    # Documented in monorepo/doc/pal/PalAdvancedProgrammingFunctions.md
    def rq_set_conveyor_clearance(is_left_pallet, height):
      if height < 0:
        popup("rq_set_conveyor_clearance(): The clearance height should be positive.", title="Palletizer", error=True,
        blocking=True)
      elif height == 0:
        height = 0.0001
      end

      pallet_side = "right"
      if(is_left_pallet):
         pallet_side = "left"
      end

      local palletId = node_rpc_server.getPalletId(pallet_side)
      node_rpc_server.setConveyorVerticalClearance(palletId, height)
    end
    ###############################################################
    # Linear Axis Move related methods
    ###############################################################
    def verify_is_in_linear_axis_range(target_axis_position):
      axis_position_range = node_rpc_server.linearaxisgetpositionrange()

      if target_axis_position < axis_position_range[0] or target_axis_position > axis_position_range[1]:
        textmsg("Linear axis target position : ", target_axis_position)
        textmsg("Linear axis position range : ", axis_position_range)
        popup("Linear axis position is unreachable.", "Linear Axis Move", blocking=True, error=True)
        halt
      end
    end

    # Documented in monorepo/doc/pal/PalAdvancedProgrammingFunctions.md
    def rq_get_linear_axis_pos():
        axis_position = node_rpc_server.linearaxisgetactualposition()
        return axis_position
    end

  BLOW_OFF_MODE_NO_AIR = 0
  BLOW_OFF_MODE_SMART_AIR = 1
  UNDEFINED_THREAD_ID = -1
  MODBUS_TYPE = "MODBUS"
  STANDARD_TYPE = "STANDARD"
  INVALID_OUTPUT_ADDRESS = -1
  RQ_UNUSED_TIMEOUT = -1

  global rq_cnc_insertion_node_ids = [-1, -1]
  global rq_run_timeout = 30

  ###################################################################################
  #
  # Generic methods
  #
  ###################################################################################

  def bool_to_str(value):
    if value:
      return "true"
    else:
      return "false"
    end
  end

  def bool_array_to_string(array, index):
    if (index >= length(array)):
      return "]"
    end

    separator = ","
    if (index == length(array) - 1):
      separator = ""
    end

    if (index == 0):
      str_array = concat("[", bool_to_str(array[index]), separator)
      return str_cat(str_array, bool_array_to_string(array, index + 1))
    else:
      return concat(bool_to_str(array[index]), separator, bool_array_to_string(array, index + 1))
    end
  end

  def rq_bool_array_to_string(array):
    return bool_array_to_string(array, 0)
  end

  def json_force_node(force, max_negative_deviation, max_positive_deviation, stiffness, enabled_axis, feature, is_adaptive):
    json = "{"
    json = concat(json, key_val("forceFrame", feature), ",")
    json = concat(json, key_val("isAdaptive", is_adaptive), ",")
    json = concat(json, key_val("isForceControlAboutActualPosition", "false"), ",")
    json = concat(json, key_val("isForceMode", enabled_axis), ",")
    json = concat(json, key_val("maxNegativeDeviation", max_negative_deviation), ",")
    json = concat(json, key_val("maxPositiveDeviation", max_positive_deviation), ",")
    json = concat(json, key_val("stiffness", stiffness), ",")
    json = concat(json, key_val("targetTcpWrench", force), "}")
    return json
  end

  def rq_setup_machine_tending_force_node(feature, force, stiffness, max_negative_deviation, max_positive_deviation, enabled_axis, is_adaptive):
    force_node_id = node_rpc_server.createnewforcenode()
    node_rpc_server.fromjson(force_node_id, json_force_node(force, max_negative_deviation, max_positive_deviation,
    stiffness, rq_bool_array_to_string(enabled_axis), 1, bool_to_str(is_adaptive)))
    return force_node_id
  end

  ###################################################################################
  #
  # TRAJECTORY UTILITIES
  #
  ###################################################################################

  def dot_product(v1, v2):
    return [v1]*transpose(v2)
  end

  def get_symmetric_poses_from_middle(p1, p2, middle_pose, distance):
    distance_p1_middle = point_dist(p1, middle_pose)
    alpha = (distance / 2) / distance_p1_middle
    start_pose = interpolate_pose(middle_pose, p1, alpha)
    end_pose = interpolate_pose(middle_pose, p2, alpha)

    return [start_pose, end_pose]
  end

  def translate_to_origin(pose):
    return p[0, 0, 0, pose[3], pose[4], pose[5]]
  end


  ###################################################################################
  #
  # ROBOTIQ PART PRESENTER
  #
  ###################################################################################

  global cnc_part_presenter_index = 0

  def rq_pallet_get_poses_from_index(p_corner_1_approach, p_corners, nb_rows, nb_columns, alternate_direction, index):
      row = floor(index / nb_columns)
      column = index % nb_columns

      row_alpha = 0
      if(nb_rows > 1):
          row_alpha = row / (nb_rows - 1)
      end

      p_row_start = interpolate_pose(p_corners[0], p_corners[3], row_alpha)
      p_row_end = interpolate_pose(p_corners[1], p_corners[2], row_alpha)

      column_alpha = 0
      if(nb_columns > 1):
          column_alpha = column / (nb_columns - 1)
      end

      if(alternate_direction and (row % 2) and nb_columns > 1):
          pallet_pose = interpolate_pose(p_row_end, p_row_start, column_alpha)
      else:
          pallet_pose = interpolate_pose(p_row_start, p_row_end, column_alpha)
      end

      T_1approach_1 = pose_trans(inv(p_corner_1_approach), p_corners[0])
      approach_pose = pose_trans(pallet_pose, inv(T_1approach_1))

      return [approach_pose, pallet_pose]
  end

  ###################################################################################
  #
  # MOVE DOOR
  #
  ###################################################################################

  def rq_setup_door_force_node(reference_frame, force, stiffness):
    feature = 1
    forces = [force,0,0,0,0,0]
    max_negative_deviation = [-5, 0, 0, 0, 0, 0]
    max_positive_deviation = [0.01, 0, 0, 0, 0, 0] # using a large value here would allow the trajectory to violate the kinematics limits, using zero removes the force node effect
    stiffnesses = [stiffness, 100, 100, 100, 100, 100]
    enabled_axis = [True, False, False, False, False, False]
    is_adaptive = True

    force_node_id = rq_setup_machine_tending_force_node(feature, forces, stiffnesses, max_negative_deviation,
    max_positive_deviation, enabled_axis, is_adaptive)

    node_rpc_server.setCustomFixedForceFrame(force_node_id, [reference_frame[3],reference_frame[4],reference_frame[5]])

    return force_node_id
  end

  def json_rq_moves_node(tcp_speed, tcp_accel):
    json = "{"
    json = concat(json, key_val("offsetType", 0), ",")
    json = concat(json, key_val("tcpSpeed", tcp_speed), ",")
    json = concat(json, key_val("tcpAccel", tcp_accel), ",")
    json = concat(json, key_val("actualreferenceframe", [0, 0, 0, 0, 0, 0]), ",")
    json = concat(json, key_val("originalreferenceframe", [0, 0, 0, 0, 0, 0]), "}")
    return json
  end

  def rq_setup_rqmoves_node(parent_node_id, tcp_speed, tcp_accel):
    rq_moves_node_id = node_rpc_server.createnewrqmoves()
    node_rpc_server.fromjson(rq_moves_node_id, json_rq_moves_node(tcp_speed, tcp_accel))
    node_rpc_server.setparentid(rq_moves_node_id, parent_node_id)
    return rq_moves_node_id
  end

  def rq_setup_waypoint_node(pose, joints, is_straight, parent_node_id):
    def json_waypoint_node(pose, joints, is_straight):
      json = "{"
      json = concat(json, key_val("jointPositions", joints), ",")
      json = concat(json, key_val("tcpPose", [pose[0],pose[1],pose[2],pose[3],pose[4],pose[5]]), ",")
      json = concat(json, key_val("isStraight", bool_to_str(is_straight)), "}")
      return json
    end

    waypoint_node_id = node_rpc_server.createnewwaypointnode()
    node_rpc_server.fromjson(waypoint_node_id, json_waypoint_node(pose, joints, is_straight))
    node_rpc_server.setparentid(waypoint_node_id, parent_node_id)
    node_rpc_server.rqmovesaddwaypoint(parent_node_id, waypoint_node_id)
    return waypoint_node_id
  end

  def rq_setup_move_door(reference_frame, start_pose, start_joints, stop_pose, stop_joints, move_force, contact_force, tcp_speed=0.4, tcp_accel=0.4):

    stop_pose_in_start_frame = pose_trans(pose_inv(start_pose), stop_pose)

    seeks_contact = False
    stiffness = 10
    move_force_node_id = rq_setup_door_force_node(reference_frame, move_force, stiffness)
    rq_moves_node_id = rq_setup_rqmoves_node(move_force_node_id, tcp_speed, tcp_accel)
    waypoint_open = rq_setup_waypoint_node(start_pose, start_joints, False, rq_moves_node_id)
    waypoint_close = rq_setup_waypoint_node(stop_pose, stop_joints, True, rq_moves_node_id)
    seeks_contact = True
    stiffness = 100
    contact_force_node_id = rq_setup_door_force_node(reference_frame, contact_force, stiffness)

    rq_movej_node_id = node_rpc_server.createnewmovejnode()
    node_rpc_server.setparentid(rq_movej_node_id, move_force_node_id)

    return [move_force_node_id, rq_moves_node_id, waypoint_open, waypoint_close, contact_force_node_id, rq_movej_node_id]
  end

  def rq_move_door(start_pose, start_joints, stop_pose, stop_joints, move_force, contact_force, tcp_speed, tcp_accel, approach_pose, approach_joints, end_reached_threshold=0.001):

    reference_frame = list_to_pose(kinematics_rpc_server.reorientP1WithXTowardP2andZApproxP1Z(start_pose, stop_pose))

    node_ids = rq_setup_move_door(reference_frame, start_pose, start_joints, stop_pose, stop_joints, move_force, contact_force, tcp_speed, tcp_accel)

    move_force_node_id = node_ids[0]
    rq_moves_node_id = node_ids[1]
    start_waypoint_node_id = node_ids[2]
    end_waypoint_node_id = node_ids[3]
    contact_force_node_id = node_ids[4]
    rq_movej_node_id = node_ids[5]

    rq_wait_ft_sensor_steady(2000)
    zero_ftsensor()
    sleep(0.1)

    path_answer = node_rpc_server.rqmovesinit(rq_moves_node_id)
    verify_path_answer(path_answer)

    approach_position_joints = get_inverse_kin(approach_pose, qnear=approach_joints)
    movej(approach_position_joints)

    node_rpc_server.movejdefinewaypoint(rq_movej_node_id, get_actual_joint_positions(), 1.0, 1.0)
    node_rpc_server.setparentid(rq_movej_node_id, move_force_node_id)
    reset_node_executor()
    active_and_reset_node(move_force_node_id)
    node_execution_thread = execute_node(rq_movej_node_id, True)

    path_answer = node_rpc_server.rqmovesinit(rq_moves_node_id)
    verify_path_answer(path_answer)
    q0 = node_rpc_server.rqmovesgetfirstpoint(rq_moves_node_id)
    node_rpc_server.setparentid(rq_movej_node_id, move_force_node_id)
    node_rpc_server.movejdefinewaypoint(rq_movej_node_id, q0, 1.0, 0.4)
    execute_node(rq_movej_node_id)
    execute_node(start_waypoint_node_id)
    execute_node(end_waypoint_node_id)

    kill_thread(node_execution_thread)

    node_rpc_server.movejdefinewaypoint(rq_movej_node_id, get_actual_joint_positions(), 1.0, 1.0)
    node_rpc_server.setparentid(rq_movej_node_id, contact_force_node_id)
    reset_node_executor()
    active_and_reset_node(contact_force_node_id)
    node_execution_thread = execute_node(rq_movej_node_id, True)

    timeout = 20
    while (point_dist(get_actual_tcp_pose(), stop_pose) > end_reached_threshold):
      if (timeout <= 0):
        popup("Door has not reached its final position")
        halt
      else:
        sync()
        timeout = timeout - get_steptime()
      end
    end

    kill_thread(node_execution_thread)

    approach_pose_in_start_frame = pose_trans(pose_inv(start_pose), approach_pose)
    retract_pose = pose_trans(get_actual_tcp_pose(), approach_pose_in_start_frame)
    movej(retract_pose)

    node_rpc_server.deletenode(move_force_node_id)
    node_rpc_server.deletenode(rq_moves_node_id)
    node_rpc_server.deletenode(start_waypoint_node_id)
    node_rpc_server.deletenode(end_waypoint_node_id)
    node_rpc_server.deletenode(contact_force_node_id)
    node_rpc_server.deletenode(rq_movej_node_id)

  end

  ###################################################################################
  #
  # CNC Insertion
  #
  ###################################################################################

  def rq_collet_insertion(contact_pose, insert_pose, inserted_pose):
      movel(contact_pose, a=1.2, v=0.025)
      movel(insert_pose, a=1.2, v=0.025)

      zero_ftsensor()
      sleep(0.1)

      direction = "Z+"
      stop_force_threshold = 3.0
      max_radius = 5.0
      radius_incr = 0.7
      peck_mode = False
      tangential_speed = 0.02
      compliant_insert_force_threshold = 10.0
      spiral_initial_pose_offset_name = "spiral_initial_pose_offset_name"
      rq_ins_destination = inserted_pose
      max_distance = point_dist(inserted_pose, get_actual_tcp_pose())
      rq_spiral_not_completed = False
      rq_ins_speed_setting = 0.02

      rq_insert_spiral_urcap(direction, stop_force_threshold, max_radius, radius_incr, peck_mode, tangential_speed, compliant_insert_force_threshold, spiral_initial_pose_offset_name)

      if (rq_spiral_not_completed):
        return False
      end

      return True
  end

  def rq_push_part(approach_pose, chuck_pose):
      zero_ftsensor()
      sleep(0.1)

      # Find pose with z axis pointing in the direction of the insertion
      p1 = translate_to_origin(approach_pose)
      insertion_dir_in_base_frame = pose_trans(p1, pose_trans(pose_inv(approach_pose), chuck_pose))
      ref_frame_pose = list_to_pose(kinematics_rpc_server.poseFromZaxis([insertion_dir_in_base_frame[0], insertion_dir_in_base_frame[1], insertion_dir_in_base_frame[2]]))

      surface_found = rq_linear_search_custom_frame("Z+", 10.0, 0.025, 0.1, ref_frame_pose)

      if not(surface_found):
          return False
      end

      return True
  end

  def rq_place_in_chuck(close_chuck_do, open_chuck_do, chuck_approach, chuck_position, chuck_delay):
      rq_open_workholding(close_chuck_do, open_chuck_do)

      movel(chuck_approach, a=1.2, v=0.25)
      movel(chuck_position, a=1.2, v=0.25)

      rq_close_workholding(close_chuck_do, open_chuck_do)
      sleep(chuck_delay)
  end

  def rq_pre_pick_in_chuck(chuck_approach, chuck_position, speed=0.25, accel=1.2):
      movel(chuck_approach, accel, speed)
      movel(chuck_position, accel, speed)
  end

  def rq_post_pick_in_chuck(close_chuck_do, open_chuck_do, chuck_approach, chuck_position, chuck_delay, speed=0.25,
  accel=1.2):
      rq_open_workholding(close_chuck_do, open_chuck_do)
      sleep(chuck_delay)

      movel(chuck_approach, accel, speed)
  end

  def rq_open_workholding(close_do, open_do):
      rq_set_workholding_do(close_do, open_do, False)
  end

  def rq_close_workholding(close_do, open_do):
      rq_set_workholding_do(close_do, open_do, True)
  end

  def rq_set_workholding_do(close_do, open_do, close_request):
      is_close_do_valid = rq_is_do_valid(close_do)
      is_open_do_valid = rq_is_do_valid(open_do)

      if(is_close_do_valid):
          set_standard_digital_out(close_do, close_request)
      end
      if(is_open_do_valid):
          set_standard_digital_out(open_do, not close_request)
      end
      if(is_close_do_valid or is_open_do_valid):
          sleep(0.5)
      end
  end

  def rq_is_do_valid(do_id):
      return do_id >= 0 and do_id <= 7
  end

  def set_cleaning_digital_output(address, state, blow_off_mode, output_type):
     if(blow_off_mode == BLOW_OFF_MODE_SMART_AIR):
       rq_set_output(output_type, address, state)
     end
  end

  ###################################################################################
  #
  # PATH GENERATOR 6 POINTS CURVE BUILT WITH 2 POINTS
  #
  ###################################################################################

  def execute_half_pipe(pose_1, pose_2,pose_transformation_air_nozzle_to_actual_tcp, depth, length_distance, width, angle, speed, spacing, address, output_type, blow_off_mode, passes):
    path_gen_poses = get_path_generator_6_points_poses(pose_1, pose_2, pose_transformation_air_nozzle_to_actual_tcp, depth, length_distance, width, angle)
    start_pose = p[path_gen_poses[0,0],path_gen_poses[0,1],path_gen_poses[0,2],path_gen_poses[0,3],path_gen_poses[0,4],path_gen_poses[0,5]]
    path_generator_node_id = setup_path_generator_6_points(path_gen_poses, speed, spacing)
    execute_path_generator_6_points(path_generator_node_id, start_pose,  address, output_type, blow_off_mode, passes)
  end

  def get_path_generator_6_points_poses(pose_2, pose_5,pose_transformation_air_nozzle_to_actual_tcp, depth=0.01, length=0, width=0.05, angle_deg=0):

    def offset_pose(pose, offset, offset_reference_frame, pose_transformation_air_nozzle_to_actual_tcp):
      pose_relative_to_ref_frame = express_pose_A_relative_to_pose_B(pose, offset_reference_frame)
      ref_frame_with_offset = pose_trans(offset_reference_frame, offset)
      pose_with_offset = pose_trans(ref_frame_with_offset, pose_relative_to_ref_frame)
      pose_with_offset_for_actual_tcp = pose_trans(pose_with_offset, pose_transformation_air_nozzle_to_actual_tcp)
      return pose_to_list(pose_with_offset_for_actual_tcp)
    end

    if(length > 0):
      middle_pose = interpolate_pose(pose_2, pose_5, 0.5)

      poses = get_symmetric_poses_from_middle(pose_2, pose_5, middle_pose, length)
      pose_2 = poses[0]
      pose_5 = poses[1]
    end

    path_ref_frame = list_to_pose(kinematics_rpc_server.reorientP1WithXTowardP2andZApproxP1Z(pose_2, pose_5))

    offset1 = pose_add(p[0,0,0,0,d2r(angle_deg),0], p[0, width,-depth,-d2r(angle_deg),0,0])
    offset2 = pose_add(p[0,0,0,0,d2r(angle_deg),0], p[0,     0,     0,              0,0,0])
    offset3 = pose_add(p[0,0,0,0,d2r(angle_deg),0], p[0,-width,-depth, d2r(angle_deg),0,0])

    pose_1_array = offset_pose(pose_2, offset1, path_ref_frame, pose_transformation_air_nozzle_to_actual_tcp)
    pose_2_array = offset_pose(pose_2, offset2, path_ref_frame, pose_transformation_air_nozzle_to_actual_tcp)
    pose_3_array = offset_pose(pose_2, offset3, path_ref_frame, pose_transformation_air_nozzle_to_actual_tcp)

    pose_4_array = offset_pose(pose_5, offset1, path_ref_frame, pose_transformation_air_nozzle_to_actual_tcp)
    pose_5_array = offset_pose(pose_5, offset2, path_ref_frame, pose_transformation_air_nozzle_to_actual_tcp)
    pose_6_array = offset_pose(pose_5, offset3, path_ref_frame, pose_transformation_air_nozzle_to_actual_tcp)

    return [pose_1_array, pose_2_array, pose_3_array, pose_4_array, pose_5_array, pose_6_array]
  end

  def setup_path_generator_6_points(pose_list, tcp_speed=0.1, spacing=0.02):

    def json_path_generator_node(pose_list, tcp_speed, spacing):

      SIX_POINTS_CURVE = 3
      OFFSET_TYPE_NONE = 0
      FORCE_OPPOSITE_SIDE = 2

      json = "{"
      json = concat(json, key_val("tcpSpeed", tcp_speed), ",")
      json = concat(json, key_val("poses", pose_list), ",")
      json = concat(json, key_val("avoidAbruptEnd", "false"), ",")
      json = concat(json, key_val("isSurfaceFillOn", "true"), ",")
      json = concat(json, key_val("spacing", spacing), ",")
      json = concat(json, key_val("pathType", SIX_POINTS_CURVE), ",")
      json = concat(json, key_val("offsetType",OFFSET_TYPE_NONE), ",")
      json = concat(json, key_val("endingMode", FORCE_OPPOSITE_SIDE), "}")

      return json
    end

    rq_path_generator_parent_id = 0
    path_generator_node_id = node_rpc_server.createPathGeneratorNode()
    node_rpc_server.fromjson(path_generator_node_id, json_path_generator_node(pose_list, tcp_speed, spacing))
    node_rpc_server.setparentid(path_generator_node_id, rq_path_generator_parent_id)

    return path_generator_node_id
  end

  def execute_path_generator_6_points(path_generator_node_id, pose_1, address = INVALID_OUTPUT_ADDRESS, output_type = MODBUS_TYPE, blow_off_mode = BLOW_OFF_MODE_NO_AIR, passes = 1):
    index = 0
    while (index < passes):
      movej(get_inverse_kin(pose_1))
      set_cleaning_digital_output(address, True, blow_off_mode, output_type)
      reset_node_executor()
      node_execution_thread = execute_node(path_generator_node_id, True)
      rq_continue_node_execution = False
      set_cleaning_digital_output(address, False, blow_off_mode, output_type)
      join node_execution_thread
      index = index + 1
    end
    node_rpc_server.deletenode(path_generator_node_id)
  end

  ###################################################################################
  #
  # Straight line trajectory
  #
  ###################################################################################

  def execute_straight_line(p1, p2,pose_transformation_air_nozzle_to_actual_tcp, accel=1.2, speed=0.25, distance = 0, angles = [0, 0, 0], address = INVALID_OUTPUT_ADDRESS, output_type = MODBUS_TYPE, blow_off_mode = BLOW_OFF_MODE_NO_AIR, passes = 1):
    offset_for_angles = p[0, 0, 0, d2r(angles[0]), d2r(angles[1]), d2r(angles[2])]
    p1 = pose_trans(p1, offset_for_angles)
    p2 = pose_trans(p2, offset_for_angles)

    # apply transformation to take into account that the actual tcp offset is not the same as the one that was used when the waypoints were saved:
    p1 = pose_trans(p1, pose_transformation_air_nozzle_to_actual_tcp)
    p2 = pose_trans(p2, pose_transformation_air_nozzle_to_actual_tcp)
    global air_output_adress = address

    qActual = get_actual_joint_positions()
    CleanPathId = node_rpc_server.createnewcleaningpathnode(p1, p2, qActual, passes, distance, accel, speed, blow_off_mode)

    reset_node_executor()
    if output_type == MODBUS_TYPE:
      air_thread = run modbusAirControlThread()
    elif output_type == STANDARD_TYPE:
      air_thread = run standardAirControlThread()
    end

    node_execution_thread = execute_node(CleanPathId, True)
    rq_continue_node_execution = False

    join node_execution_thread
    node_rpc_server.deletenode(CleanPathId)
    if output_type == MODBUS_TYPE or output_type == STANDARD_TYPE :
      kill air_thread
    end
  end

  ###################################################################################
  #
  # Cross trajectory
  #
  ###################################################################################

  def find_cross_trajectory_poses(p1, p2, height=0, width=0, p1_angles = [0, 0, 0], p2_angles = [0, 0, 0], p3_angles = [0, 0, 0], p4_angles = [0, 0, 0]):
    def find_side_poses(p0, p1):
      def find_side_pose(p0,p1,angle):
        p1_T_p0 = pose_trans(pose_inv(p0), p1)
        rotated_p0_by_90_degrees = pose_trans(p0, p[0, 0, 0, 0, 0, d2r(angle)])

        side_pose = pose_trans(rotated_p0_by_90_degrees, p1_T_p0)
        side_pose[3] = p0[3]
        side_pose[4] = p0[4]
        side_pose[5] = p0[5]

        return side_pose
      end

      p3= find_side_pose(p0, p1, 90)
      p4 = find_side_pose(p0, p1, 270)

      return [p3, p4]
    end

    def get_start_and_end_poses_based_on_distance(p1, p2, middle_pose, distance):
      if(distance == 0):
        start_pose = p1
        end_pose = p2
      else:
        poses = get_symmetric_poses_from_middle(p1, p2, middle_pose, distance)
        start_pose = poses[0]
        end_pose = poses[1]
      end
      return [start_pose, end_pose]
    end

    def get_side_poses_based_on_distance(p1, p2, middle_pose, width):
      if(width == 0):
        side_poses = find_side_poses(middle_pose, p1)
      else:
        poses = get_symmetric_poses_from_middle(p1, p2, middle_pose, width)
        side_poses = find_side_poses(middle_pose, poses[0])
      end

      return side_poses
    end

    def get_angle_offset(angles):
      return  p[0, 0, 0, d2r(angles[0]), d2r(angles[1]), d2r(angles[2])]
    end

    middle_pose = interpolate_pose(p1, p2, 0.5)

    start_and_end_poses = get_start_and_end_poses_based_on_distance(p1, p2, middle_pose, height)
    side_poses = get_side_poses_based_on_distance(p1, p2, middle_pose, width)

    p1_offset = get_angle_offset(p1_angles)
    p2_offset = get_angle_offset(p2_angles)
    p3_offset = get_angle_offset(p3_angles)
    p4_offset = get_angle_offset(p4_angles)

    start_and_end_poses[0] = pose_trans(start_and_end_poses[0], p1_offset)
    start_and_end_poses[1] = pose_trans(start_and_end_poses[1], p2_offset)
    side_poses[0] = pose_trans(side_poses[0], p3_offset)
    side_poses[1] = pose_trans(side_poses[1], p4_offset)

    return [middle_pose, start_and_end_poses[0], start_and_end_poses[1], side_poses[0], side_poses[1]]
  end

  def execute_cross_trajectory(p1, p2,pose_transformation_air_nozzle_to_actual_tcp, height=0, width=0, p1_angles = [0, 0, 0], p2_angles = [0, 0, 0], p3_angles = [0, 0, 0], p4_angles = [0, 0, 0], accel=1.2, speed=0.25,  address = INVALID_OUTPUT_ADDRESS, output_type = MODBUS_TYPE, blow_off_mode = BLOW_OFF_MODE_NO_AIR, passes = 1):

    cross_poses = find_cross_trajectory_poses(p1, p2, height, width, p1_angles, p2_angles, p3_angles, p4_angles)

    p0 = pose_trans(cross_poses[0], pose_transformation_air_nozzle_to_actual_tcp)
    p1 = pose_trans(cross_poses[1], pose_transformation_air_nozzle_to_actual_tcp)
    p2 = pose_trans(cross_poses[2], pose_transformation_air_nozzle_to_actual_tcp)
    p3 = pose_trans(cross_poses[3], pose_transformation_air_nozzle_to_actual_tcp)
    p4 = pose_trans(cross_poses[4], pose_transformation_air_nozzle_to_actual_tcp)

   index = 0

   while (index < passes):
     movej(get_inverse_kin(p0))
     set_cleaning_digital_output(address, True, blow_off_mode, output_type)
     movel(p1, accel, speed)
     movel(p2, accel, speed)
     movel(p0, accel, speed)
     movel(p3, accel, speed)
     movel(p4, accel, speed)
     set_cleaning_digital_output(address, False, blow_off_mode, output_type)
     index = index + 1
   end
  end

  def execute_waypoint_cross_trajectory(starting_pose, finishing_pose, accel=1.2, speed=0.25):
   movej(get_inverse_kin(starting_pose))
   movel(finishing_pose, accel, speed)
  end

  ###################################################################################
  #
  # Fermat spiral trajectory
  #
  ###################################################################################

  def execute_fermat_spiral(start_pose, end_pose,pose_transformation_air_nozzle_to_actual_tcp, max_radius = 0, angle = 0, number_of_turns = 1, speed = 0.25,address = INVALID_OUTPUT_ADDRESS, output_type = MODBUS_TYPE, blow_off_mode = BLOW_OFF_MODE_NO_AIR, passes = 1):
    def find_middle(start_pose, end_pose):
      alpha = 0.5
      return interpolate_pose(start_pose, end_pose, alpha)
    end

    def find_next_theta(spiral_constant, theta, speed):
      denom = spiral_constant * sqrt(1/(4*theta) + theta)
      theta_dot = speed / denom
      theta = theta + theta_dot * rq_controller_time_step
      return theta
    end

    def find_spiral_pose(theta, spiral_plane, center_pose, angle, spiral_constant, pose_transformation_air_nozzle_to_actual_tcp):
      local r = spiral_constant * sqrt(theta)
      local x = r * cos(theta)
      local y = r * sin(theta)

      local p2 = pose_trans(spiral_plane, p[x,y,0,0,0,0])
      local p3 = p[p2[0], p2[1], p2[2], center_pose[3], center_pose[4], center_pose[5]]
      local p4 = pose_trans(p3, pose_transformation_air_nozzle_to_actual_tcp)
      local p5 = pose_trans(p4, p[0, 0, 0, -d2r(angle)*cos(theta), -d2r(angle)*sin(theta), 0])
      return p5
    end

    def execute_outer_to_inner_spiral(start_pose, middle_pose, spiral_plane, pose_transformation_air_nozzle_to_actual_tcp, max_angle, angle, spiral_constant_nominal, speed, address, output_type, blow_off_mode):
      local theta = max_angle
      local max_r = point_dist(start_pose, middle_pose)
      local spiral_constant = -1 * spiral_constant_nominal
      local r = max_r
      local is_first_pose = True

      while (norm((r)) <= max_r):
        theta = find_next_theta(spiral_constant, theta, speed)
        if(theta < 0):
          break
        end

        r = spiral_constant * sqrt(theta)
        next_pose = find_spiral_pose(theta, spiral_plane, middle_pose, angle, spiral_constant, pose_transformation_air_nozzle_to_actual_tcp)

        if (is_first_pose):
          movej(get_inverse_kin(next_pose))
          set_cleaning_digital_output(address, True, blow_off_mode, output_type)
          is_first_pose = False
        else:
          servoj(get_inverse_kin(next_pose), t = rq_controller_time_step)
        end
      end
    end

    def execute_inner_to_outer_spiral(start_pose, middle_pose, spiral_plane, pose_transformation_air_nozzle_to_actual_tcp, angle, spiral_constant, speed):
      local theta = 0.0001
      local max_r = point_dist(start_pose, middle_pose)
      local r = 0

      while (norm(r) <= max_r):
        theta = find_next_theta(spiral_constant, theta, speed)
        r = spiral_constant * sqrt(theta)
        next_pose = find_spiral_pose(theta, spiral_plane, middle_pose, angle, spiral_constant, pose_transformation_air_nozzle_to_actual_tcp)
        servoj(get_inverse_kin(next_pose), t = rq_controller_time_step)
      end
    end

    max_angle = d2r(number_of_turns * 360)
    middle_pose = find_middle(start_pose, end_pose)

    if(max_radius > 0):
      poses = get_symmetric_poses_from_middle(start_pose, end_pose, middle_pose, max_radius * 2)
      start_pose = poses[0]
      end_pose = poses[1]
    end

    SPIRAL_CONSTANT = (point_dist(middle_pose, start_pose)) / sqrt(max_angle)

    spiral_plane = list_to_pose(kinematics_rpc_server.reorientP1WithXTowardP2andZApproxP1Z(middle_pose, end_pose))


    index = 0
    while(index < passes):
      execute_outer_to_inner_spiral(start_pose, middle_pose, spiral_plane,pose_transformation_air_nozzle_to_actual_tcp, max_angle, angle, SPIRAL_CONSTANT, speed, address, output_type, blow_off_mode)
      execute_inner_to_outer_spiral(end_pose, middle_pose, spiral_plane, pose_transformation_air_nozzle_to_actual_tcp, angle, SPIRAL_CONSTANT, speed)
      set_cleaning_digital_output(address, False, blow_off_mode, output_type)
      index = index + 1
    end
  end

  ###################################################################################
  #
  # ROBOTIQ VISE INSERTION
  #
  # - The first touch is performed in the direction of the gravity, regardless of
  #   the robot mounting orientation, tcp offset and TCP orientation
  # - Optional 2e et 3e touch are performed relative to TCP. They require that, at
  #   the moment that the insertion is performed, the TCP is oriented such that one
  #   axis is aligned with the gravity. The TCP axes for the 2e and 3e touch are
  #   chosen as the ones not aligned with the gravity.
  ###################################################################################
  def insert_in_vise(start_pose, end_pose, number_of_touch=3, forces=[10, 20, 20], invert_axis=False, move_to_end_pose=False):

    def list_by_scalar_multiply_(l1, scalar):
      result = l1
      i=0
      while i<length(result):
        result[i]=l1[i]*scalar
        i=i+1
      end
      return result
    end

    def find_gravity_direction(acceleration_direction, threshold):
      result = [False, False, False]
      i = 0
      while i < length(result):
        result[i] =  norm(acceleration_direction[i]) > threshold
        i = i + 1
      end
      return result
    end

    def get_axis(index, direction):
      axis = "XYZ"
      if direction < 0:
        sign = "-"
      elif direction > 0:
        sign = "+"
      else:
        popup("insert_in_vise:get_axis >>> direction cannot be 0. Fix it.")
        halt
      end
      return str_cat(str_sub(axis, index, 1), sign)
    end

    def direction_to_index(str):
      if "X" == str_sub(str, 0, 1):
        return 0
      elif "Y" == str_sub(str, 0, 1):
        return 1
      elif "Z" == str_sub(str, 0, 1):
        return 2
      else:
        popup("invalid direction :", str)
        halt
      end
    end

    def find_touch_direction(mask, direction):
      i = 0
      result = [0, 0, 0]
      while i < 3:
        if mask[i]:
          result[i] = direction[i]
        end
        i = i + 1
      end
      return result
    end

    def find_touch_direction_str(mask, direction):
      i = 0
      result = ""
      while i < 3:
        if mask[i]:
          result = str_cat(result, get_axis(i, direction[i]))
        end
        i = i + 1
      end
      return result
    end

    def invert(list):
      result = list
      i = 0
      while i < length(list):
        result[i] = not list[i]
        i = i + 1
      end
      return result
    end

    def assert_that_the_first_touch_is_aligned_with_an_axis(first_touch_direction_mask):
      i = 0
      counter = 0
      while i < length(first_touch_direction_mask):
        if first_touch_direction_mask[i]:
          counter = counter + 1
        end
        i = i + 1
      end

      if counter != 1:
        popup("One of the TCP axes must be perpendicular to the floor while loading the part in the vise.")
        halt
      end
    end

    def setup_nodes(forces, number_of_touch, first_touch_direction_mask, direction, second_direction_str, third_direction_str):
      def max_deviation_from(forces, enabled_axis):
        i = 0
        deviation = [0, 0, 0, 0, 0, 0]
        while i < 3:
          if forces[i] > 0:
            deviation[i] = 10
          elif forces[i] ==  0:
            deviation[i] = 10
          end
          i = i + 1
        end
        while i < 6:
          if enabled_axis[i]:
            deviation[i] = 0.35
          end
          i = i + 1
        end
        return deviation
      end

      def min_deviation_from(forces, enabled_axis):
        i = 0
        deviation = [0, 0, 0, 0, 0, 0]
        while i < 3:
          if forces[i] < 0:
            deviation[i] = -10
          elif forces[i] ==  0:
            deviation[i] = -10
          end
          i = i + 1
        end
        while i < 6:
          if enabled_axis[i]:
            deviation[i] = -0.35
          end
          i = i + 1
        end
        return deviation
      end

      def stiffness_from(forces):
        i = 0
        stiffness = [0, 0, 0, 100, 100, 100]
        while i < length(forces):
          if norm(forces[i]) > 0:
            stiffness[i] = 100
          else:
            stiffness[i] = 85
          end
          i = i + 1
        end
        return stiffness
      end

      def compute_final_forces(forces, number_of_touch, first_touch_direction_mask, direction, second_direction_str, third_direction_str):
        final_forces = [0, 0, 0]
        if number_of_touch > 0:
          i = 0
          while i < length(first_touch_direction_mask):
            if first_touch_direction_mask[i]:
              break
            end
            i = i + 1
          end
          final_forces[i] = direction[i] * forces[i]
        end
        if number_of_touch > 1:
          i = direction_to_index(second_direction_str)
          final_forces[i] = direction[i] * forces[i]
        end
        if number_of_touch > 2:
          i = direction_to_index(third_direction_str)
          final_forces[i] = direction[i] * forces[i]
        end
        return final_forces
      end

      def compute_enabled_axis(first_touch_direction_mask):
        enabled_axis = [True, True, True, False, False, False]
        i = 0
        while i < length(first_touch_direction_mask):
          if first_touch_direction_mask[i]:
            break
          end
          i = i + 1
        end
        enabled_axis[i + 3] = True

        return enabled_axis
      end

      final_forces = compute_final_forces(forces, number_of_touch, first_touch_direction_mask, direction, second_direction_str, third_direction_str)
      enabled_axis = compute_enabled_axis(first_touch_direction_mask)

      force_node_id = rq_setup_machine_tending_force_node(1, [final_forces[0], final_forces[1], final_forces[2], 0, 0, 0], stiffness_from
      (final_forces), min_deviation_from(final_forces, enabled_axis), max_deviation_from(final_forces, enabled_axis),
      enabled_axis, False)
      movej_node_id = node_rpc_server.createnewmovejnode()
      node_rpc_server.setparentid(movej_node_id, force_node_id)

      return [force_node_id, movej_node_id]
    end

    def average_tool_acceleration_reading(n_samples, delay):
      n = n_samples
      reading = [0, 0, 0]
      while n > 0:
        reading = reading + get_tool_accelerometer_reading()
        sleep(delay)
        n = n - 1
      end
      return reading/n_samples
    end

    def linear_search_toward_gravity(force):
      # maybe add a stopj here to prevent acceleration reading to be influenced by robot movement
      flange_accel = average_tool_acceleration_reading(10, 0.1) # measured accel is oriented in gravity oposite direction
      flange_accel_pose = p[-flange_accel[0], -flange_accel[1], -flange_accel[2], 0, 0,0]
      p1 = translate_to_origin(get_actual_tool_flange_pose())
      gravity_dir_in_base_frame = pose_trans(p1, flange_accel_pose)

      # Find pose with z axis pointing in gravity direction:
      ref_frame_pose = list_to_pose(kinematics_rpc_server.poseFromZaxis([gravity_dir_in_base_frame[0], gravity_dir_in_base_frame[1], gravity_dir_in_base_frame[2]]))
      speed = 0.01
      abs_max_distance = 0.05

      surface_found = rq_linear_search_custom_frame("Z+", force, speed, abs_max_distance, ref_frame_pose)
      return surface_found
    end

    #### Actual insert_in_vise method ####
    movel(start_pose)
    zero_ftsensor()

    # 1. Use accelerometer reading to find touches directions:
    ACCELERATION_THRESHOLD = 8
    flange_accel = average_tool_acceleration_reading(10, 0.1)
    tcp_accel = pose_trans(pose_inv(get_tcp_offset()), p[flange_accel[0], flange_accel[1], flange_accel[2], 0, 0, 0])
    first_touch_direction_mask = find_gravity_direction(tcp_accel, ACCELERATION_THRESHOLD)
    assert_that_the_first_touch_is_aligned_with_an_axis(first_touch_direction_mask)

    direction_transform = pose_trans(pose_inv(start_pose), end_pose)
    direction = [direction_transform[0], direction_transform[1], direction_transform[2]]
    direction_sign = [direction[0]/norm(direction[0]), direction[1]/norm(direction[1]), direction[2]/norm(direction[2])]

    touch_direction_str = find_touch_direction_str(invert(first_touch_direction_mask), direction_sign)
    touch_direction = find_touch_direction(invert(first_touch_direction_mask), direction_sign)

    if invert_axis:
      second_direction_str = str_sub(touch_direction_str, 0, 2)
      third_direction_str = str_sub(touch_direction_str, 2, 4)
    else:
      second_direction_str = str_sub(touch_direction_str, 2, 4)
      third_direction_str = str_sub(touch_direction_str, 0, 2)
    end

    end_pose_orientation = translate_to_origin(end_pose)

    # 2. Prepare nodes:
    rq_cnc_insertion_node_ids = setup_nodes(forces, number_of_touch, first_touch_direction_mask, direction_sign, second_direction_str, third_direction_str)
    feature_tool = 1

    # 3. Perform touches:
    if number_of_touch > 0:
      surface_found = linear_search_toward_gravity(forces[0])
      if not surface_found:
        textmsg("Insertion in vise: First contact has not been found")
        popup("First contact has not been found", title="Insertion in vise", blocking=True)
        return UNDEFINED_THREAD_ID
      end
    end
    if number_of_touch > 1:
      surface_found = rq_linear_search_urcap(second_direction_str, forces[1], 0.01, 0.05, feature_tool)
      if not surface_found:
        textmsg("Insertion in vise: Second contact has not been found")
        popup("Second contact has not been found", title="Insertion in vise", blocking=True)
        return UNDEFINED_THREAD_ID
      end
    end
    if number_of_touch > 2:
      surface_found = rq_linear_search_urcap(third_direction_str, forces[2], 0.01, 0.05, feature_tool)
      if not surface_found:
        textmsg("Insertion in vise: Third contact has not been found")
        popup("Third contact has not been found", title="Insertion in vise", blocking=True)
        return UNDEFINED_THREAD_ID
      end
    end

    # 4. Move to end position:
    if not move_to_end_pose:
      end_pose = get_actual_tcp_pose()
    end

    node_rpc_server.movejdefinewaypoint(rq_cnc_insertion_node_ids[1], get_actual_joint_positions(), 1.0, 1.0)
    reset_node_executor()
    active_and_reset_node(rq_cnc_insertion_node_ids[0])
    node_execution_thread = execute_node(rq_cnc_insertion_node_ids[1], True)
    node_rpc_server.movejdefinewaypoint(rq_cnc_insertion_node_ids[1], get_inverse_kin(end_pose), 1.0, 1.0)
    execute_node(rq_cnc_insertion_node_ids[1])
    sleep(1)
    return node_execution_thread
  end

  ###################################################################################
  # AIR OUTPUT CONTROL
  ###################################################################################
  thread modbusAirControlThread():
    while (True):
      rq_air_value = read_input_boolean_register(101)
      modbus_set_output_signal(air_output_adress, rq_air_value, False)
      sleep(rq_controller_time_step)
    end
  end

  thread standardAirControlThread():
    while (True):
      rq_air_value = read_input_boolean_register(101)
      set_digital_out(air_output_adress, rq_air_value)
      sleep(rq_controller_time_step)
    end
  end
  def rq_set_output(output_type, address, value):
    if output_type == "MODBUS":
      modbus_set_output_signal(address, value)
    elif output_type == "STANDARD":
      set_standard_digital_out(address, value)
    end
  end

  def rq_digital_output_action(action, output_type, address, time_on=1, time_off=0.5, delay_after=0):
    if action == "PUSH_AND_HOLD":
      rq_set_output(output_type, address, True)
    elif action == "PUSH":
      rq_set_output(output_type, address, True)
      sleep(time_on)
      rq_set_output(output_type, address, False)
    elif action == "DOUBLE_PUSH":
      rq_set_output(output_type, address, True)
      sleep(time_on)
      rq_set_output(output_type, address, False)
      sleep(time_off)
      rq_set_output(output_type, address, True)
      sleep(time_on)
      rq_set_output(output_type, address, False)
    elif action == "RELEASE":
      rq_set_output(output_type, address, False)
    end
    sleep(delay_after)
  end
  def json_kinematic_parameters_ratio(ratio):
    json = "{"
    json = concat(json, key_val("kinematicParametersRatio", ratio), "}")
    return json
  end

  def execute_move_along_trail(trail_node_id, joint_positions, kinematic_parameters_ratio):
    node_rpc_server.fromjson(trail_node_id, json_kinematic_parameters_ratio(kinematic_parameters_ratio))
    roadmap_state = node_rpc_server.initRoadmap(trail_node_id, joint_positions)
    path_time = roadmap_state[0]

    if(path_time > 0.0):
      reset_node_executor()
      node_execution_thread = execute_node(trail_node_id, True)
      kill node_execution_thread
    end
  end
    global servojId = 2
  rq_collision_detection_stop()
  # end: URCap Installation Node
  global timer_1=0
  global c2_p=p[-.028463494537, -.307727419006, .173332682584, -3.141059388184, -.056193760799, -.000004272450]
  global c2_q=[-1.2244494597064417, -1.496974529033043, -1.7373507022857666, -1.4773324069431801, 1.5717664957046509, 3.4508044719696045]
  global s2_p=p[-.028856690118, -.249726646426, .145170222541, 3.141026680054, .055975812019, -.000017180394]
  global s2_q=[-1.1368125120746058, -1.2298501592925568, -2.0743727684020996, -1.4073492002538224, 1.5715453624725342, 3.5388050079345703]
  global c1_p=p[.079726385078, -.307004063818, .173197835475, -3.141081840863, -.055829763070, .000000336873]
  global c1_q=[-0.8901303450213831, -1.5340925504318257, -1.703249454498291, -1.4742992383292695, 1.571800947189331, 3.7853426933288574]
  global s1_p=p[.079339633526, -.249019256999, .138958933641, -3.141083724909, -.056146777813, .000021861818]
  global s1_q=[-0.736511532460348, -1.2886369985393067, -2.066201686859131, -1.3568056237748642, 1.5716667175292969, 3.9390151500701904]
  global chipC_p=p[-.099700577098, -.183627440197, .208433402457, 3.139691259007, -.105394058226, -.000149781669]
  global chipC_q=[-1.3891781012164515, -1.0096948903850098, -1.88504958152771, -1.8167749843993128, 1.5708818435668945, 3.388993501663208]
  global Waypoint_25_p=p[-.122879871442, -.368965239733, .188211838452, 3.139821275232, -.105433326911, -.000075080205]
  global Waypoint_25_q=[-1.5479124228106897, -1.8512498341002406, -1.271846055984497, -1.5885349712767542, 1.5719534158706665, 3.2300467491149902]
  global Waypoint_26_p=p[-.293995928019, -.360529248638, .222497263242, 3.139820833490, -.105446172100, -.000068418500]
  global Waypoint_26_q=[-1.9689658323871058, -2.3604399166502894, -0.28896433115005493, -2.062209268609518, 1.571913719177246, 2.8087823390960693]
  global Waypoint_27_p=p[-.293996037589, -.360524548960, .073401623062, -3.139818121402, .105463968189, .000065100461]
  global Waypoint_27_q=[-1.9687660376178187, -2.2716170750060023, -1.1700339317321777, -1.2699676317027588, 1.5726664066314697, 2.809603691101074]
  global Waypoint_28_p=p[-.293994929318, -.360517570897, .073396573982, -3.079220194370, .622813891331, .000072005146]
  global Waypoint_28_q=[-1.9687660376177893, -2.2716089687261967, -1.1700649262597302, -1.269964114900139, 1.572658061981124, 3.141592653589793]
  global Waypoint_29_p=p[-.293994178547, -.360515134427, .073402631236, -3.140584062493, .078656845609, .000054923880]
  global Waypoint_29_q=[-1.9687698523153152, -2.2715932331392654, -1.1700625419823325, -1.2699834567121284, 1.5726652145390896, 2.792526803190927]
  global Waypoint_30_p=p[-.293991359760, -.360511345669, .073405660262, -3.079212155022, .622831433047, .000021425167]
  global Waypoint_30_q=[-1.9687779585452905, -2.271581312216341, -1.170064806944243, -1.2700025898209706, 1.5726886987653534, 3.141592653589793]
  global Waypoint_31_p=p[-.293995928019, -.360529248638, .222497263242, 3.139820833490, -.105446172100, -.000068418500]
  global Waypoint_31_q=[-1.9689658323871058, -2.3604399166502894, -0.28896433115005493, -2.062209268609518, 1.571913719177246, 2.8087823390960693]
  global Waypoint_32_p=p[-.120064390322, -.465070651334, .187365924664, 2.700279766902, -.088400420341, .019763045538]
  global Waypoint_32_q=[-1.5412524382220667, -1.9475652180113734, -1.406833291053772, -0.9173591893962403, 1.5603561401367188, 3.2332537174224854]
  global Waypoint_33_p=p[-.125099110421, -.299097154487, .189878767902, 3.139750209928, -.105401717856, -.000111797080]
  global Waypoint_33_q=[-1.550074879323141, -1.5617311683348198, -1.5979981422424316, -1.5518303674510499, 1.5716702938079834, 3.2279696464538574]
  global Waypoint_1_p=p[.263501689877, -.337317763427, .239349489480, 3.139797243720, -.105347053477, -.000037720516]
  global Waypoint_1_q=[-0.5959728399859827, -2.1057659588255824, -0.6533136367797852, -1.9525557957091273, 1.5718059539794922, 4.181682586669922]
  global Waypoint_2_p=p[.265438435610, -.352444474661, .141740907029, 3.139726376264, -.105360108121, -.000022031768]
  global Waypoint_2_q=[-0.6231134573565882, -2.1016999683775843, -1.126999020576477, -1.4828875821879883, 1.5722739696502686, 4.154912948608398]
  global Waypoint_3_p=p[.206441973084, -.349241721273, .141737893294, 3.139734184252, -.105329347268, -.000022485776]
  global Waypoint_3_q=[-0.7073677221881312, -1.9410401783385218, -1.3681066036224365, -1.4024366003325959, 1.5721865892410278, 4.070710182189941]
  global Waypoint_4_p=p[.157616611756, -.378012026932, .141738203587, 3.139764187573, -.105376653239, -.000076760662]
  global Waypoint_4_q=[-0.8494070211993616, -1.9579774341978968, -1.3439116477966309, -1.409730003481247, 1.5722019672393799, 3.928692579269409]
  global Waypoint_5_p=p[.109134761588, -.393436595889, .141742225598, 3.139732501163, -.105376381431, -.000050533951]
  global Waypoint_5_q=[-0.972816292439596, -1.9523960552611292, -1.3519116640090942, -1.4072665137103577, 1.5721949338912964, 3.805286407470703]
  global Waypoint_6_p=p[-.188131250090, -.345166366147, .141750553976, 3.139727051239, -.105353578209, -.000024875816]
  global Waypoint_6_q=[-1.7293437162982386, -1.8864180050291957, -1.4439769983291626, -1.381135032778122, 1.572224736213684, 3.0487747192382812]
  global Waypoint_7_p=p[-.131564048097, -.216205376465, .141741700579, 3.139714533984, -.105382776464, -.000044168049]
  global Waypoint_7_q=[-1.572542969380514, -1.2417927545360108, -2.0833356380462646, -1.3863917154124756, 1.571577787399292, 3.2058310508728027]
  global timer_1_is_counting=False
  thread Timer_Thread():
    while (True):
      if (timer_1_is_counting):
        timer_1 = timer_1 + get_steptime()
      end
      sync()
    end
  end
  run Timer_Thread()
  def CircleAllangles_1():
    $ 156 "CircleAllangles_1" "noBreak"
    $ 157 "r≔25/1000"
    global r=25/1000
    $ 158 "A≔31"
    global A=31
    $ 159 "A≔A*3.1416/180"
    global A=A*3.1416/180
    $ 160 "p0≔p[c[0]-r,c[1],c[2],c[3],c[4],c[5]-1.5*A]"
    global p0=p[c[0]-r,c[1],c[2],c[3],c[4],c[5]-1.5*A]
    $ 161 "p45≔p[c[0]-0.71*r,c[1]+0.71*r,c[2],c[3]-A/1.1,c[4],c[5]-A/1.1]"
    global p45=p[c[0]-0.71*r,c[1]+0.71*r,c[2],c[3]-A/1.1,c[4],c[5]-A/1.1]
    $ 162 "p90≔p[c[0],c[1]+r,c[2],c[3]-A,c[4],c[5]]"
    global p90=p[c[0],c[1]+r,c[2],c[3]-A,c[4],c[5]]
    $ 163 "p135≔p[c[0]+0.71*r,c[1]+0.71*r,c[2],c[3]-A/1.1,c[4],c[5]+A/1.1]"
    global p135=p[c[0]+0.71*r,c[1]+0.71*r,c[2],c[3]-A/1.1,c[4],c[5]+A/1.1]
    $ 164 "p180≔p[c[0]+r,c[1],c[2],c[3],c[4],c[5]+1.5*A]"
    global p180=p[c[0]+r,c[1],c[2],c[3],c[4],c[5]+1.5*A]
    $ 165 "p225≔p[c[0]+0.71*r,c[1]-0.71*r,c[2],c[3]+A/1.1,c[4],c[5]+A/1.1]"
    global p225=p[c[0]+0.71*r,c[1]-0.71*r,c[2],c[3]+A/1.1,c[4],c[5]+A/1.1]
    $ 166 "p270≔p[c[0],c[1]-r,c[2],c[3]+A,c[4],c[5]]"
    global p270=p[c[0],c[1]-r,c[2],c[3]+A,c[4],c[5]]
    $ 167 "p315≔p[c[0]-0.71*r,c[1]-0.71*r,c[2],c[3]+A/1.1,c[4],c[5]-A/1.1]"
    global p315=p[c[0]-0.71*r,c[1]-0.71*r,c[2],c[3]+A/1.1,c[4],c[5]-A/1.1]
    $ 168 "Set atomization=On"
    set_standard_digital_out(1, True)
    $ 169 "Set triggersolenoid=On"
    set_standard_digital_out(0, True)
    $ 170 "MoveL"
    $ 171 "p0" "breakAfter"
    set_tcp(p[0.0,0.0,0.11,0.0,0.0,0.0])
    movel(p0, a=1.2, v=0.12, r=0.01)
    $ 172 "p45" "breakAfter"
    set_tcp(p[0.0,0.0,0.11,0.0,0.0,0.0])
    movel(p45, a=1.2, v=0.12, r=0.01)
    $ 173 "p90" "breakAfter"
    set_tcp(p[0.0,0.0,0.11,0.0,0.0,0.0])
    movel(p90, a=1.2, v=0.12, r=0.01)
    $ 174 "p135" "breakAfter"
    set_tcp(p[0.0,0.0,0.11,0.0,0.0,0.0])
    movel(p135, a=1.2, v=0.12, r=0.01)
    $ 175 "p180" "breakAfter"
    set_tcp(p[0.0,0.0,0.11,0.0,0.0,0.0])
    movel(p180, a=1.2, v=0.12, r=0.01)
    $ 176 "Set triggersolenoid=Off"
    set_standard_digital_out(0, False)
    $ 177 "Wait: 0.1"
    sleep(0.1)
    $ 178 "Set triggersolenoid=On"
    set_standard_digital_out(0, True)
    $ 179 "p225" "breakAfter"
    set_tcp(p[0.0,0.0,0.11,0.0,0.0,0.0])
    movel(p225, a=1.2, v=0.12, r=0.01)
    $ 180 "p270" "breakAfter"
    set_tcp(p[0.0,0.0,0.11,0.0,0.0,0.0])
    movel(p270, a=1.2, v=0.12, r=0.01)
    $ 181 "p315" "breakAfter"
    set_tcp(p[0.0,0.0,0.11,0.0,0.0,0.0])
    movel(p315, a=1.2, v=0.12, r=0.01)
    $ 182 "p0" "breakAfter"
    set_tcp(p[0.0,0.0,0.11,0.0,0.0,0.0])
    movel(p0, a=1.2, v=0.12, r=0.01)
    $ 183 "p45" "breakAfter"
    set_tcp(p[0.0,0.0,0.11,0.0,0.0,0.0])
    movel(p45, a=1.2, v=0.12, r=0.01)
    $ 184 "Set triggersolenoid=Off"
    set_standard_digital_out(0, False)
    $ 185 "Wait: 0.1"
    sleep(0.1)
    $ 186 "Set triggersolenoid=On"
    set_standard_digital_out(0, True)
    $ 187 "p90" "breakAfter"
    set_tcp(p[0.0,0.0,0.11,0.0,0.0,0.0])
    movel(p90, a=1.2, v=0.12, r=0.01)
    $ 188 "p135" "breakAfter"
    set_tcp(p[0.0,0.0,0.11,0.0,0.0,0.0])
    movel(p135, a=1.2, v=0.12, r=0.01)
    $ 189 "p180" "breakAfter"
    set_tcp(p[0.0,0.0,0.11,0.0,0.0,0.0])
    movel(p180, a=1.2, v=0.12, r=0.01)
    $ 190 "p225" "breakAfter"
    set_tcp(p[0.0,0.0,0.11,0.0,0.0,0.0])
    movel(p225, a=1.2, v=0.12, r=0.01)
    $ 191 "Set triggersolenoid=Off"
    set_standard_digital_out(0, False)
    $ 192 "Wait: 0.1"
    sleep(0.1)
    $ 193 "Set triggersolenoid=On"
    set_standard_digital_out(0, True)
    $ 194 "p270" "breakAfter"
    set_tcp(p[0.0,0.0,0.11,0.0,0.0,0.0])
    movel(p270, a=1.2, v=0.12, r=0.01)
    $ 195 "p315" "breakAfter"
    set_tcp(p[0.0,0.0,0.11,0.0,0.0,0.0])
    movel(p315, a=1.2, v=0.12, r=0.01)
    $ 196 "p0" "breakAfter"
    set_tcp(p[0.0,0.0,0.11,0.0,0.0,0.0])
    movel(p0, a=1.2, v=0.12, r=0.01)
    $ 197 "Set triggersolenoid=Off"
    set_standard_digital_out(0, False)
    $ 198 "Wait: 0.1"
    sleep(0.1)
    $ 199 "Set atomization=Off"
    set_standard_digital_out(1, False)
  end
  def Spraychip2():
    $ 200 "Spraychip2" "noBreak"
    $ 201 "MoveJ"
    $ 202 "chipC" "breakAfter"
    movej(get_inverse_kin(chipC_p, qnear=chipC_q), a=1.3962634015954636, v=1.0471975511965976)
    $ 203 "c≔chipC"
    global c=chipC_p
    $ 204 "rc≔27/1000"
    global rc=27/1000
    $ 205 "p0≔p[c[0]+rc,c[1],c[2],c[3],c[4],c[5]-1.5*0]"
    global p0=p[c[0]+rc,c[1],c[2],c[3],c[4],c[5]-1.5*0]
    $ 206 "p45≔p[c[0]+0.71*rc,c[1]+0.71*rc,c[2],c[3]-0/1.1,c[4],c[5]-0/1.1]"
    global p45=p[c[0]+0.71*rc,c[1]+0.71*rc,c[2],c[3]-0/1.1,c[4],c[5]-0/1.1]
    $ 207 "p90≔p[c[0],c[1]+rc,c[2],c[3]-0,c[4],c[5]]"
    global p90=p[c[0],c[1]+rc,c[2],c[3]-0,c[4],c[5]]
    $ 208 "p135≔p[c[0]-0.71*rc,c[1]+0.71*rc,c[2],c[3]-0/1.1,c[4],c[5]+0/1.1]"
    global p135=p[c[0]-0.71*rc,c[1]+0.71*rc,c[2],c[3]-0/1.1,c[4],c[5]+0/1.1]
    $ 209 "p180≔p[c[0]-rc,c[1],c[2],c[3],c[4],c[5]+1.5*0]"
    global p180=p[c[0]-rc,c[1],c[2],c[3],c[4],c[5]+1.5*0]
    $ 210 "p225≔p[c[0]-0.71*rc,c[1]-0.71*rc,c[2],c[3]+0/1.1,c[4],c[5]+0/1.1]"
    global p225=p[c[0]-0.71*rc,c[1]-0.71*rc,c[2],c[3]+0/1.1,c[4],c[5]+0/1.1]
    $ 211 "p270≔p[c[0],c[1]-rc,c[2],c[3]+0,c[4],c[5]]"
    global p270=p[c[0],c[1]-rc,c[2],c[3]+0,c[4],c[5]]
    $ 212 "p315≔p[c[0]+0.71*rc,c[1]-0.71*rc,c[2],c[3]+0/1.1,c[4],c[5]-0/1.1]"
    global p315=p[c[0]+0.71*rc,c[1]-0.71*rc,c[2],c[3]+0/1.1,c[4],c[5]-0/1.1]
    $ 213 "Set atomization=On"
    set_standard_digital_out(1, True)
    $ 214 "Set triggersolenoid=On"
    set_standard_digital_out(0, True)
    $ 215 "MoveL"
    $ 216 "p0" "breakAfter"
    set_tcp(p[0.0,0.0,0.11,0.0,0.0,0.0])
    movel(p0, a=1.3, v=0.07, r=0.01)
    $ 217 "p45" "breakAfter"
    set_tcp(p[0.0,0.0,0.11,0.0,0.0,0.0])
    movel(p45, a=1.3, v=0.07, r=0.01)
    $ 218 "p90" "breakAfter"
    set_tcp(p[0.0,0.0,0.11,0.0,0.0,0.0])
    movel(p90, a=1.3, v=0.07, r=0.01)
    $ 219 "p135" "breakAfter"
    set_tcp(p[0.0,0.0,0.11,0.0,0.0,0.0])
    movel(p135, a=1.3, v=0.07, r=0.01)
    $ 220 "p180" "breakAfter"
    set_tcp(p[0.0,0.0,0.11,0.0,0.0,0.0])
    movel(p180, a=1.3, v=0.07, r=0.01)
    $ 221 "Set triggersolenoid=Off"
    set_standard_digital_out(0, False)
    $ 222 "Wait: 0.1"
    sleep(0.1)
    $ 223 "Set triggersolenoid=On"
    set_standard_digital_out(0, True)
    $ 224 "p225" "breakAfter"
    set_tcp(p[0.0,0.0,0.11,0.0,0.0,0.0])
    movel(p225, a=1.3, v=0.07, r=0.01)
    $ 225 "p270" "breakAfter"
    set_tcp(p[0.0,0.0,0.11,0.0,0.0,0.0])
    movel(p270, a=1.3, v=0.07, r=0.01)
    $ 226 "p315" "breakAfter"
    set_tcp(p[0.0,0.0,0.11,0.0,0.0,0.0])
    movel(p315, a=1.3, v=0.07, r=0.01)
    $ 227 "p0" "breakAfter"
    set_tcp(p[0.0,0.0,0.11,0.0,0.0,0.0])
    movel(p0, a=1.3, v=0.07, r=0.01)
    $ 228 "p45" "breakAfter"
    set_tcp(p[0.0,0.0,0.11,0.0,0.0,0.0])
    movel(p45, a=1.3, v=0.07, r=0.01)
    $ 229 "Set triggersolenoid=Off"
    set_standard_digital_out(0, False)
    $ 230 "Wait: 0.1"
    sleep(0.1)
    $ 231 "Set triggersolenoid=On"
    set_standard_digital_out(0, True)
    $ 232 "p90" "breakAfter"
    set_tcp(p[0.0,0.0,0.11,0.0,0.0,0.0])
    movel(p90, a=1.3, v=0.07, r=0.01)
    $ 233 "p135" "breakAfter"
    set_tcp(p[0.0,0.0,0.11,0.0,0.0,0.0])
    movel(p135, a=1.3, v=0.07, r=0.01)
    $ 234 "p180" "breakAfter"
    set_tcp(p[0.0,0.0,0.11,0.0,0.0,0.0])
    movel(p180, a=1.3, v=0.07, r=0.01)
    $ 235 "p225" "breakAfter"
    set_tcp(p[0.0,0.0,0.11,0.0,0.0,0.0])
    movel(p225, a=1.3, v=0.07, r=0.01)
    $ 236 "p270" "breakAfter"
    set_tcp(p[0.0,0.0,0.11,0.0,0.0,0.0])
    movel(p270, a=1.3, v=0.07, r=0.01)
    $ 237 "p315" "breakAfter"
    set_tcp(p[0.0,0.0,0.11,0.0,0.0,0.0])
    movel(p315, a=1.3, v=0.07, r=0.01)
    $ 238 "p0" "breakAfter"
    set_tcp(p[0.0,0.0,0.11,0.0,0.0,0.0])
    movel(p0, a=1.3, v=0.07, r=0.01)
    $ 239 "MoveJ"
    $ 241 "chipC" "breakAfter"
    movej(get_inverse_kin(chipC_p, qnear=chipC_q), a=1.3962634015954636, v=1.0471975511965976)
    $ 242 "Wait: 0.2"
    sleep(0.2)
    $ 243 "Set triggersolenoid=Off"
    set_standard_digital_out(0, False)
    $ 244 "Wait: 0.1"
    sleep(0.1)
    $ 245 "Set atomization=Off"
    set_standard_digital_out(1, False)
  end
  def spray2():
    $ 246 "spray2" "noBreak"
    $ 247 "r≔45/1000"
    global r=45/1000
    $ 248 "A≔0"
    global A=0
    $ 249 "p0≔p[c[0]-r,c[1],c[2],c[3],c[4],c[5]-1.5*A]"
    global p0=p[c[0]-r,c[1],c[2],c[3],c[4],c[5]-1.5*A]
    $ 250 "p45≔p[c[0]-0.71*r,c[1]+0.71*r,c[2],c[3]-A/1.1,c[4],c[5]-A/1.1]"
    global p45=p[c[0]-0.71*r,c[1]+0.71*r,c[2],c[3]-A/1.1,c[4],c[5]-A/1.1]
    $ 251 "p90≔p[c[0],c[1]+r,c[2],c[3]-A,c[4],c[5]]"
    global p90=p[c[0],c[1]+r,c[2],c[3]-A,c[4],c[5]]
    $ 252 "p135≔p[c[0]+0.71*r,c[1]+0.71*r,c[2],c[3]-A/1.1,c[4],c[5]+A/1.1]"
    global p135=p[c[0]+0.71*r,c[1]+0.71*r,c[2],c[3]-A/1.1,c[4],c[5]+A/1.1]
    $ 253 "p180≔p[c[0]+r,c[1],c[2],c[3],c[4],c[5]+1.5*A]"
    global p180=p[c[0]+r,c[1],c[2],c[3],c[4],c[5]+1.5*A]
    $ 254 "p225≔p[c[0]+0.71*r,c[1]-0.71*r,c[2],c[3]+A/1.1,c[4],c[5]+A/1.1]"
    global p225=p[c[0]+0.71*r,c[1]-0.71*r,c[2],c[3]+A/1.1,c[4],c[5]+A/1.1]
    $ 255 "p270≔p[c[0],c[1]-r,c[2],c[3]+A,c[4],c[5]]"
    global p270=p[c[0],c[1]-r,c[2],c[3]+A,c[4],c[5]]
    $ 256 "p315≔p[c[0]-0.71*r,c[1]-0.71*r,c[2],c[3]+A/1.1,c[4],c[5]-A/1.1]"
    global p315=p[c[0]-0.71*r,c[1]-0.71*r,c[2],c[3]+A/1.1,c[4],c[5]-A/1.1]
    $ 257 "Set atomization=On"
    set_standard_digital_out(1, True)
    $ 258 "Set triggersolenoid=On"
    set_standard_digital_out(0, True)
    $ 259 "MoveL"
    $ 260 "p0" "breakAfter"
    set_tcp(p[0.0,0.0,0.11,0.0,0.0,0.0])
    movel(p0, a=1.2, v=0.12, r=0.01)
    $ 261 "p45" "breakAfter"
    set_tcp(p[0.0,0.0,0.11,0.0,0.0,0.0])
    movel(p45, a=1.2, v=0.12, r=0.01)
    $ 262 "p90" "breakAfter"
    set_tcp(p[0.0,0.0,0.11,0.0,0.0,0.0])
    movel(p90, a=1.2, v=0.12, r=0.01)
    $ 263 "p135" "breakAfter"
    set_tcp(p[0.0,0.0,0.11,0.0,0.0,0.0])
    movel(p135, a=1.2, v=0.12, r=0.01)
    $ 264 "p180" "breakAfter"
    set_tcp(p[0.0,0.0,0.11,0.0,0.0,0.0])
    movel(p180, a=1.2, v=0.12, r=0.01)
    $ 265 "Set triggersolenoid=Off"
    set_standard_digital_out(0, False)
    $ 266 "Wait: 0.1"
    sleep(0.1)
    $ 267 "Set triggersolenoid=On"
    set_standard_digital_out(0, True)
    $ 268 "p225" "breakAfter"
    set_tcp(p[0.0,0.0,0.11,0.0,0.0,0.0])
    movel(p225, a=1.2, v=0.12, r=0.01)
    $ 269 "p270" "breakAfter"
    set_tcp(p[0.0,0.0,0.11,0.0,0.0,0.0])
    movel(p270, a=1.2, v=0.12, r=0.01)
    $ 270 "p315" "breakAfter"
    set_tcp(p[0.0,0.0,0.11,0.0,0.0,0.0])
    movel(p315, a=1.2, v=0.12, r=0.01)
    $ 271 "p0" "breakAfter"
    set_tcp(p[0.0,0.0,0.11,0.0,0.0,0.0])
    movel(p0, a=1.2, v=0.12, r=0.01)
    $ 272 "p45" "breakAfter"
    set_tcp(p[0.0,0.0,0.11,0.0,0.0,0.0])
    movel(p45, a=1.2, v=0.12, r=0.01)
    $ 273 "Set triggersolenoid=Off"
    set_standard_digital_out(0, False)
    $ 274 "Wait: 0.1"
    sleep(0.1)
    $ 275 "Set triggersolenoid=On"
    set_standard_digital_out(0, True)
    $ 276 "p90" "breakAfter"
    set_tcp(p[0.0,0.0,0.11,0.0,0.0,0.0])
    movel(p90, a=1.2, v=0.12, r=0.01)
    $ 277 "p135" "breakAfter"
    set_tcp(p[0.0,0.0,0.11,0.0,0.0,0.0])
    movel(p135, a=1.2, v=0.12, r=0.01)
    $ 278 "p180" "breakAfter"
    set_tcp(p[0.0,0.0,0.11,0.0,0.0,0.0])
    movel(p180, a=1.2, v=0.12, r=0.01)
    $ 279 "p225" "breakAfter"
    set_tcp(p[0.0,0.0,0.11,0.0,0.0,0.0])
    movel(p225, a=1.2, v=0.12, r=0.01)
    $ 280 "Set triggersolenoid=Off"
    set_standard_digital_out(0, False)
    $ 281 "Wait: 0.1"
    sleep(0.1)
    $ 282 "Set triggersolenoid=On"
    set_standard_digital_out(0, True)
    $ 283 "p270" "breakAfter"
    set_tcp(p[0.0,0.0,0.11,0.0,0.0,0.0])
    movel(p270, a=1.2, v=0.12, r=0.01)
    $ 284 "p315" "breakAfter"
    set_tcp(p[0.0,0.0,0.11,0.0,0.0,0.0])
    movel(p315, a=1.2, v=0.12, r=0.01)
    $ 285 "p0" "breakAfter"
    set_tcp(p[0.0,0.0,0.11,0.0,0.0,0.0])
    movel(p0, a=1.2, v=0.12, r=0.01)
    $ 286 "Set triggersolenoid=Off"
    set_standard_digital_out(0, False)
    $ 287 "Wait: 0.1"
    sleep(0.1)
    $ 288 "Set atomization=Off"
    set_standard_digital_out(1, False)
  end
  def cleaning():
    $ 313 "cleaning" "noBreak"
    $ 314 "MoveJ"
    $ 315 "Waypoint_25" "breakAfter"
    movej(get_inverse_kin(Waypoint_25_p, qnear=Waypoint_25_q), a=1.3962634015954636, v=1.0471975511965976)
    $ 316 "Waypoint_26" "breakAfter"
    movej(get_inverse_kin(Waypoint_26_p, qnear=Waypoint_26_q), a=1.3962634015954636, v=1.0471975511965976)
    $ 317 "Waypoint_27" "breakAfter"
    movej(get_inverse_kin(Waypoint_27_p, qnear=Waypoint_27_q), a=1.3962634015954636, v=1.0471975511965976)
    $ 318 "Waypoint_28" "breakAfter"
    movej(get_inverse_kin(Waypoint_28_p, qnear=Waypoint_28_q), a=1.3962634015954636, v=1.0471975511965976)
    $ 319 "Waypoint_29" "breakAfter"
    movej(get_inverse_kin(Waypoint_29_p, qnear=Waypoint_29_q), a=1.3962634015954636, v=1.0471975511965976)
    $ 320 "Waypoint_30" "breakAfter"
    movej(get_inverse_kin(Waypoint_30_p, qnear=Waypoint_30_q), a=1.3962634015954636, v=1.0471975511965976)
    $ 321 "Waypoint_31" "breakAfter"
    movej(get_inverse_kin(Waypoint_31_p, qnear=Waypoint_31_q), a=1.3962634015954636, v=1.0471975511965976)
    $ 322 "Waypoint_32" "breakAfter"
    movej(get_inverse_kin(Waypoint_32_p, qnear=Waypoint_32_q), a=1.3962634015954636, v=1.0471975511965976)
    $ 323 "Set atomization=On"
    set_standard_digital_out(1, True)
    $ 324 "Set triggersolenoid=On"
    set_standard_digital_out(0, True)
    $ 325 "Wait: 0.2"
    sleep(0.2)
    $ 326 "Set triggersolenoid=Off"
    set_standard_digital_out(0, False)
    $ 327 "Wait: 0.1"
    sleep(0.1)
    $ 328 "Set atomization=Off"
    set_standard_digital_out(1, False)
    $ 329 "Waypoint_33" "breakAfter"
    movej(get_inverse_kin(Waypoint_33_p, qnear=Waypoint_33_q), a=1.3962634015954636, v=1.0471975511965976)
  end
  def turntable():
    $ 330 "turntable" "noBreak"
    $ 331 "MoveJ"
    $ 332 "Waypoint_1" "breakAfter"
    set_tcp(p[0.0,0.0,0.11,0.0,0.0,0.0])
    movej(get_inverse_kin(pose_trans(carouselrod, pose_trans(p[-.225374943892, -.334963115589, .194760490875, -3.139766958133, .106894280099, .000011796372], Waypoint_1_p)), qnear=Waypoint_1_q), a=1.3962634015954636, v=0.5235987755982988, r=0.02)
    $ 333 "Waypoint_2" "breakAfter"
    set_tcp(p[0.0,0.0,0.11,0.0,0.0,0.0])
    movej(get_inverse_kin(pose_trans(carouselrod, pose_trans(p[-.225374943892, -.334963115589, .194760490875, -3.139766958133, .106894280099, .000011796372], Waypoint_2_p)), qnear=Waypoint_2_q), a=1.3962634015954636, v=0.5235987755982988, r=0.02)
    $ 334 "Waypoint_3" "breakAfter"
    set_tcp(p[0.0,0.0,0.11,0.0,0.0,0.0])
    movej(get_inverse_kin(pose_trans(carouselrod, pose_trans(p[-.225374943892, -.334963115589, .194760490875, -3.139766958133, .106894280099, .000011796372], Waypoint_3_p)), qnear=Waypoint_3_q), a=1.3962634015954636, v=0.5235987755982988, r=0.02)
    $ 335 "Waypoint_4" "breakAfter"
    set_tcp(p[0.0,0.0,0.11,0.0,0.0,0.0])
    movej(get_inverse_kin(pose_trans(carouselrod, pose_trans(p[-.225374943892, -.334963115589, .194760490875, -3.139766958133, .106894280099, .000011796372], Waypoint_4_p)), qnear=Waypoint_4_q), a=1.3962634015954636, v=0.5235987755982988, r=0.02)
    $ 336 "Waypoint_5" "breakAfter"
    set_tcp(p[0.0,0.0,0.11,0.0,0.0,0.0])
    movej(get_inverse_kin(pose_trans(carouselrod, pose_trans(p[-.225374943892, -.334963115589, .194760490875, -3.139766958133, .106894280099, .000011796372], Waypoint_5_p)), qnear=Waypoint_5_q), a=1.3962634015954636, v=0.5235987755982988, r=0.02)
    $ 337 "MoveJ"
    $ 338 "Waypoint_6" "breakAfter"
    movej(get_inverse_kin(pose_trans(carouselrod, pose_trans(p[-.225374943892, -.334963115589, .194760490875, -3.139766958133, .106894280099, .000011796372], Waypoint_6_p)), qnear=Waypoint_6_q), a=1.3962634015954636, v=0.3141592653589793)
    $ 339 "Wait: 1.0"
    sleep(1.0)
    $ 340 "MoveJ"
    $ 341 "Waypoint_7" "breakAfter"
    movej(get_inverse_kin(pose_trans(carouselrod, pose_trans(p[-.225374943892, -.334963115589, .194760490875, -3.139766958133, .106894280099, .000011796372], Waypoint_7_p)), qnear=Waypoint_7_q), a=1.3962634015954636, v=1.0471975511965976, r=0.02)
  end
  def SmallTunnel():
    $ 342 "SmallTunnel" "noBreak"
    $ 343 "q1≔p[q[0],q[1],q[2]+0.05,q[3],q[4],q[4]]"
    global q1=p[q[0],q[1],q[2]+0.05,q[3],q[4],q[4]]
    $ 344 "q2≔p[q[0],q[1],q[2]+0.02,q[3],q[4],q[5]]"
    global q2=p[q[0],q[1],q[2]+0.02,q[3],q[4],q[5]]
    $ 345 "Set atomization=On"
    set_standard_digital_out(1, True)
    $ 346 "Set triggersolenoid=On"
    set_standard_digital_out(0, True)
    $ 347 "Wait: 0.05"
    sleep(0.05)
    $ 348 "Set triggersolenoid=Off"
    set_standard_digital_out(0, False)
    $ 349 "Wait: 0.1"
    sleep(0.1)
    $ 350 "Set atomization=Off"
    set_standard_digital_out(1, False)
    $ 351 "MoveL"
    $ 352 "q2" "breakAfter"
    movel(q2, a=1.2, v=0.25)
    $ 353 "Set atomization=On"
    set_standard_digital_out(1, True)
    $ 354 "Set triggersolenoid=On"
    set_standard_digital_out(0, True)
    $ 355 "q1" "breakAfter"
    movel(q1, a=1.2, v=0.25)
    $ 356 "Set triggersolenoid=Off"
    set_standard_digital_out(0, False)
    $ 357 "Wait: 0.1"
    sleep(0.1)
    $ 358 "Set atomization=Off"
    set_standard_digital_out(1, False)
  end
  while (True):
    $ 2 "Robot Program"
    $ 3 "'Program is to be used for part #127765-201 rev A telescope optical bench'"
    # 'Program is to be used for part #127765-201 rev A telescope optical bench'
    $ 4 "'Program rev ___: mm/dd/yy note'"
    # 'Program rev ___: mm/dd/yy note'
    $ 5 "timer_1: Start"
    timer_1_is_counting = True
    $ 6 "r≔25/1000"
    global r=25/1000
    $ 7 "A≔25"
    global A=25
    $ 8 "A≔A*3.1416/180"
    global A=A*3.1416/180
    $ 9 "current_coat≔1"
    global current_coat=1
    $ 10 "position≔1"
    global position=1
    $ 11 "Loop_1≔1"
    global Loop_1=1
    $ 12 "sidenum≔2"
    global sidenum=2
    $ 14 "partnum≔'Enter the number of mask sets on the carousel:'"
    global partnum=request_integer_from_primary_client("Enter the number of mask sets on the carousel:")
    $ 16 "coatnum≔'Enter the number of mask sets on the carousel:'"
    global coatnum=request_integer_from_primary_client("Enter the number of mask sets on the carousel:")
    $ 17 "If partnum≤sidenum"
    global thread_flag_17=0
    thread Thread_if_17():
      $ 18 "Loop (coatnum)>0"
      thread Thread_while_18():
        while (True):
          $ 19 "partleft≔partnum"
          global partleft=partnum
          $ 20 "loopnum≔1"
          global loopnum=1
          $ 21 "Loop partleft>0"
          thread Thread_while_21():
            while (True):
              $ 22 "If loopnum≟1"
              if (loopnum == 1):
                $ 23 "Call cleaning"
                cleaning()
                $ 24 "Call Spraychip2"
                Spraychip2()
              end
              $ 25 "If loopnum≟1 or loopnum≟3 or loopnum≟5 or loopnum≟7 or loopnum≟9 or loopnum≟11"
              global thread_flag_25=0
              thread Thread_if_25():
                $ 55 "MoveJ"
                $ 56 "c2" "breakAfter"
                movej(get_inverse_kin(c2_p, qnear=c2_q), a=1.3962634015954636, v=1.0471975511965976)
                $ 57 "c≔c2"
                global c=c2_p
                $ 58 "Call CircleAllangles_1"
                CircleAllangles_1()
                $ 59 "MoveJ"
                $ 60 "s2" "breakAfter"
                movej(get_inverse_kin(s2_p, qnear=s2_q), a=1.3962634015954636, v=1.0471975511965976)
                $ 61 "q≔s2"
                global q=s2_p
                $ 62 "Call SmallTunnel"
                SmallTunnel()
                $ 63 "MoveJ"
                $ 64 "c" "breakAfter"
                movej(c, a=1.3962634015954636, v=1.0471975511965976)
                $ 66 "position≔position+1"
                global position=position+1
                thread_flag_25 = 1
              end
              if (loopnum == 1  or  loopnum == 3  or  loopnum == 5  or  loopnum == 7  or  loopnum == 9  or  loopnum == 11):
                global thread_handler_25=run Thread_if_25()
                while (thread_flag_25 == 0):
                  if not(loopnum == 1  or  loopnum == 3  or  loopnum == 5  or  loopnum == 7  or  loopnum == 9  or  loopnum == 11):
                    kill thread_handler_25
                    thread_flag_25 = 2
                  else:
                    sync()
                  end
                end
              else:
                thread_flag_25 = 2
              end
              if (thread_flag_25 == 2):
                $ 67 "Else" "noBreak"
                $ 96 "MoveJ"
                $ 97 "c1" "breakAfter"
                movej(get_inverse_kin(c1_p, qnear=c1_q), a=1.3962634015954636, v=1.0471975511965976)
                $ 98 "c≔c1"
                global c=c1_p
                $ 99 "Call CircleAllangles_1"
                CircleAllangles_1()
                $ 100 "MoveJ"
                $ 101 "s1" "breakAfter"
                set_tcp(p[0.0,0.0,0.11,0.0,0.0,0.0])
                movej(get_inverse_kin(s1_p, qnear=s1_q), a=1.3962634015954636, v=1.0471975511965976)
                $ 102 "q≔s1"
                global q=s1_p
                $ 103 "Call SmallTunnel"
                SmallTunnel()
                $ 104 "MoveJ"
                $ 105 "c" "breakAfter"
                movej(c, a=1.3962634015954636, v=1.0471975511965976)
                $ 107 "position≔position+1"
                global position=position+1
              end
              $ 108 "loopnum≔loopnum+1"
              global loopnum=loopnum+1
              $ 109 "partleft≔partleft-1"
              global partleft=partleft-1
            end
          end
          if (partleft>0):
            global thread_handler_21=run Thread_while_21()
            while (partleft>0):
              sync()
            end
            kill thread_handler_21
          end
          $ 110 "i≔0"
          global i=0
          $ 111 "coatnum≔coatnum-1"
          global coatnum=coatnum-1
        end
      end
      if ((coatnum)>0):
        global thread_handler_18=run Thread_while_18()
        while ((coatnum)>0):
          sync()
        end
        kill thread_handler_18
      end
      $ 112 "Halt"
      halt
      thread_flag_17 = 1
    end
    if (partnum <= sidenum):
      global thread_handler_17=run Thread_if_17()
      while (thread_flag_17 == 0):
        if not(partnum <= sidenum):
          kill thread_handler_17
          thread_flag_17 = 2
        else:
          sync()
        end
      end
    else:
      thread_flag_17 = 2
    end
    if (thread_flag_17 == 2):
      $ 113 "Else" "noBreak"
      $ 114 "Loop (coatnum)>0"
      thread Thread_while_114():
        while (True):
          $ 115 "partleft≔partnum"
          global partleft=partnum
          $ 116 "loopnum≔1"
          global loopnum=1
          $ 117 "turnnum≔0"
          global turnnum=0
          $ 118 "Loop partleft>0"
          thread Thread_while_118():
            while (True):
              $ 119 "If loopnum≟1"
              if (loopnum == 1):
                $ 120 "Call cleaning"
                cleaning()
                $ 121 "Call Spraychip2"
                Spraychip2()
              end
              $ 122 "If loopnum≟1 or loopnum≟3 or loopnum≟5 or loopnum≟7 or loopnum≟9 or loopnum≟11"
              global thread_flag_122=0
              thread Thread_if_122():
                $ 123 "MoveJ"
                $ 124 "c2" "breakAfter"
                movej(get_inverse_kin(c2_p, qnear=c2_q), a=1.3962634015954636, v=1.0471975511965976)
                $ 125 "c≔c2"
                global c=c2_p
                $ 126 "Call CircleAllangles_1"
                CircleAllangles_1()
                $ 127 "MoveJ"
                $ 128 "s2" "breakAfter"
                movej(get_inverse_kin(s2_p, qnear=s2_q), a=1.3962634015954636, v=1.0471975511965976)
                $ 129 "q≔s2"
                global q=s2_p
                $ 130 "Call SmallTunnel"
                SmallTunnel()
                $ 131 "MoveJ"
                $ 132 "c" "breakAfter"
                movej(c, a=1.3962634015954636, v=1.0471975511965976)
                $ 134 "position≔position+1"
                global position=position+1
                thread_flag_122 = 1
              end
              if (loopnum == 1  or  loopnum == 3  or  loopnum == 5  or  loopnum == 7  or  loopnum == 9  or  loopnum == 11):
                global thread_handler_122=run Thread_if_122()
                while (thread_flag_122 == 0):
                  if not(loopnum == 1  or  loopnum == 3  or  loopnum == 5  or  loopnum == 7  or  loopnum == 9  or  loopnum == 11):
                    kill thread_handler_122
                    thread_flag_122 = 2
                  else:
                    sync()
                  end
                end
              else:
                thread_flag_122 = 2
              end
              if (thread_flag_122 == 2):
                $ 135 "Else" "noBreak"
                $ 136 "MoveJ"
                $ 137 "c1" "breakAfter"
                movej(get_inverse_kin(c1_p, qnear=c1_q), a=1.3962634015954636, v=1.0471975511965976)
                $ 138 "c≔c1"
                global c=c1_p
                $ 139 "Call CircleAllangles_1"
                CircleAllangles_1()
                $ 140 "MoveJ"
                $ 141 "s1" "breakAfter"
                set_tcp(p[0.0,0.0,0.11,0.0,0.0,0.0])
                movej(get_inverse_kin(s1_p, qnear=s1_q), a=1.3962634015954636, v=1.0471975511965976)
                $ 142 "q≔s1"
                global q=s1_p
                $ 143 "Call SmallTunnel"
                SmallTunnel()
                $ 144 "MoveJ"
                $ 145 "c" "breakAfter"
                movej(c, a=1.3962634015954636, v=1.0471975511965976)
                $ 147 "position≔position+1"
                global position=position+1
              end
              $ 148 "loopnum≔loopnum+1"
              global loopnum=loopnum+1
              $ 149 "partleft≔partleft-1"
              global partleft=partleft-1
            end
          end
          if (partleft>0):
            global thread_handler_118=run Thread_while_118()
            while (partleft>0):
              sync()
            end
            kill thread_handler_118
          end
          $ 150 "i≔0"
          global i=0
          $ 151 "Loop (6-turnnum)>0"
          thread Thread_while_151():
            while (True):
              $ 152 "Call turntable"
              turntable()
              $ 153 "turnnum≔turnnum+1"
              global turnnum=turnnum+1
            end
          end
          if ((6-turnnum)>0):
            global thread_handler_151=run Thread_while_151()
            while ((6-turnnum)>0):
              sync()
            end
            kill thread_handler_151
          end
          $ 154 "coatnum≔coatnum-1"
          global coatnum=coatnum-1
        end
      end
      if ((coatnum)>0):
        global thread_handler_114=run Thread_while_114()
        while ((coatnum)>0):
          sync()
        end
        kill thread_handler_114
      end
      $ 155 "Halt"
      halt
    end
  end
end
